(* IEC 61131-3 sources: sigmatek-logger-api/IXON_API/Class/cIXONConv10Value, 1 file *)

(* ---- cIXONConv10Value.st ---- *)
#DEFINE MAX_NAME_LENGTH 100
#DEFINE MAX_VALUE_LENGTH 10
#DEFINE MAX_DATASTRING_LENGTH 1024

(*!
<Class
	Name               = "cIXONConv10Value"
	Revision           = "0.0"
	RealtimeTask       = "false"
	CyclicTask         = "false"
	BackgroundTask     = "false"
	Sigmatek           = "false"
	OSInterface        = "false"
	HighPriority       = "false"
	Automatic          = "false"
	UpdateMode         = "Prescan"
	SharedCommandTable = "true"
	Objectsize         = "(510,120)">
	<Channels>
		<Server Name="ClassSvr" Visualized="false" Initialize="false" WriteProtected="true" Retentive="false"/>
		<Server Name="sCmdConvert" Visualized="false" Initialize="false" WriteProtected="false" Retentive="false"/>
		<Server Name="sName1" Class="String" Visualized="true" Initialize="true" WriteProtected="false" Retentive="false"/>
		<Server Name="sName10" Class="String" Visualized="true" Initialize="true" WriteProtected="false" Retentive="false"/>
		<Server Name="sName2" Class="String" Visualized="true" Initialize="true" WriteProtected="false" Retentive="false"/>
		<Server Name="sName3" Class="String" Visualized="true" Initialize="true" WriteProtected="false" Retentive="false"/>
		<Server Name="sName4" Class="String" Visualized="true" Initialize="true" WriteProtected="false" Retentive="false"/>
		<Server Name="sName5" Class="String" Visualized="true" Initialize="true" WriteProtected="false" Retentive="false"/>
		<Server Name="sName6" Class="String" Visualized="true" Initialize="true" WriteProtected="false" Retentive="false"/>
		<Server Name="sName7" Class="String" Visualized="true" Initialize="true" WriteProtected="false" Retentive="false"/>
		<Server Name="sName8" Class="String" Visualized="true" Initialize="true" WriteProtected="false" Retentive="false"/>
		<Server Name="sName9" Class="String" Visualized="true" Initialize="true" WriteProtected="false" Retentive="false"/>
		<Server Name="sSetInitNrOfEntrys" Visualized="false" Initialize="true" DefValue="1" WriteProtected="true" Retentive="false"/>
		<Server Name="sTriggerName" Class="String" Visualized="false" Initialize="true" WriteProtected="true" Retentive="false"/>
		<Server Name="sValue1" Visualized="false" Initialize="false" WriteProtected="false" Retentive="false"/>
		<Server Name="sValue10" Visualized="false" Initialize="false" WriteProtected="false" Retentive="false"/>
		<Server Name="sValue2" Visualized="false" Initialize="false" WriteProtected="false" Retentive="false"/>
		<Server Name="sValue3" Visualized="false" Initialize="false" WriteProtected="false" Retentive="false"/>
		<Server Name="sValue4" Visualized="false" Initialize="false" WriteProtected="false" Retentive="false"/>
		<Server Name="sValue5" Visualized="false" Initialize="false" WriteProtected="false" Retentive="false"/>
		<Server Name="sValue6" Visualized="false" Initialize="false" WriteProtected="false" Retentive="false"/>
		<Server Name="sValue7" Visualized="false" Initialize="false" WriteProtected="false" Retentive="false"/>
		<Server Name="sValue8" Visualized="false" Initialize="false" WriteProtected="false" Retentive="false"/>
		<Server Name="sValue9" Visualized="false" Initialize="false" WriteProtected="false" Retentive="false"/>
		<Client Name="Name1" Required="true" Internal="true"/>
		<Client Name="Name10" Required="true" Internal="true"/>
		<Client Name="Name2" Required="true" Internal="true"/>
		<Client Name="Name3" Required="true" Internal="true"/>
		<Client Name="Name4" Required="true" Internal="true"/>
		<Client Name="Name5" Required="true" Internal="true"/>
		<Client Name="Name6" Required="true" Internal="true"/>
		<Client Name="Name7" Required="true" Internal="true"/>
		<Client Name="Name8" Required="true" Internal="true"/>
		<Client Name="Name9" Required="true" Internal="true"/>
		<Client Name="ocSigCLib" Required="false" Internal="false"/>
		<Client Name="ToIXON_LoggerAPI" Required="true" Internal="false"/>
		<Client Name="TriggerName" Required="true" Internal="true"/>
	</Channels>
	<Separators>
		<Servers>
			<SepChn Position="3"/>
			<SepChn Position="5"/>
		</Servers>
	</Separators>
	<Network Name="cIXONConv10Value">
		<!-- List of Components in this network -->
		<Components>
			<Object
				Name       = "Name1"
				Class      = "String"
				Position   = "(420,300)"
				Visualized = "true"
				Remotely   = "true">
				<Channels>
					<Server Name="Data"/>
					<Client Name="SingleRealloc" Value="1"/>
				</Channels>
			</Object>
			<Object
				Name       = "Name10"
				Class      = "String"
				Position   = "(420,1650)"
				Visualized = "true"
				Remotely   = "true">
				<Channels>
					<Server Name="Data"/>
					<Client Name="SingleRealloc" Value="1"/>
				</Channels>
			</Object>
			<Object
				Name       = "Name2"
				Class      = "String"
				Position   = "(420,450)"
				Visualized = "true"
				Remotely   = "true">
				<Channels>
					<Server Name="Data"/>
					<Client Name="SingleRealloc" Value="1"/>
				</Channels>
			</Object>
			<Object
				Name       = "Name3"
				Class      = "String"
				Position   = "(420,600)"
				Visualized = "true"
				Remotely   = "true">
				<Channels>
					<Server Name="Data"/>
					<Client Name="SingleRealloc" Value="1"/>
				</Channels>
			</Object>
			<Object
				Name       = "Name4"
				Class      = "String"
				Position   = "(420,750)"
				Visualized = "true"
				Remotely   = "true">
				<Channels>
					<Server Name="Data"/>
					<Client Name="SingleRealloc" Value="1"/>
				</Channels>
			</Object>
			<Object
				Name       = "Name5"
				Class      = "String"
				Position   = "(420,900)"
				Visualized = "true"
				Remotely   = "true">
				<Channels>
					<Server Name="Data"/>
					<Client Name="SingleRealloc" Value="1"/>
				</Channels>
			</Object>
			<Object
				Name       = "Name6"
				Class      = "String"
				Position   = "(420,1050)"
				Visualized = "true"
				Remotely   = "true">
				<Channels>
					<Server Name="Data"/>
					<Client Name="SingleRealloc" Value="1"/>
				</Channels>
			</Object>
			<Object
				Name       = "Name7"
				Class      = "String"
				Position   = "(420,1200)"
				Visualized = "true"
				Remotely   = "true">
				<Channels>
					<Server Name="Data"/>
					<Client Name="SingleRealloc" Value="1"/>
				</Channels>
			</Object>
			<Object
				Name       = "Name8"
				Class      = "String"
				Position   = "(420,1350)"
				Visualized = "true"
				Remotely   = "true">
				<Channels>
					<Server Name="Data"/>
					<Client Name="SingleRealloc" Value="1"/>
				</Channels>
			</Object>
			<Object
				Name       = "Name9"
				Class      = "String"
				Position   = "(420,1500)"
				Visualized = "true"
				Remotely   = "true">
				<Channels>
					<Server Name="Data"/>
					<Client Name="SingleRealloc" Value="1"/>
				</Channels>
			</Object>
			<Object
				Name       = "TriggerName"
				Class      = "String"
				Position   = "(420,150)"
				Visualized = "true"
				Remotely   = "true">
				<Channels>
					<Server Name="Data"/>
					<Client Name="SingleRealloc" Value="1"/>
				</Channels>
			</Object>
		</Components>
		<Comments>
		</Comments>
		<!-- List of Connections in this network -->
		<Connections>
			<Connection Source="this.TriggerName" Destination="TriggerName.Data"/>
			<Connection Source="this.sTriggerName" Destination="TriggerName.Data" Vertices="(968,330),(796,240),"/>
			<Connection Source="this.Name1" Destination="Name1.Data"/>
			<Connection Source="this.sName1" Destination="Name1.Data" Vertices="(968,450),(796,390),"/>
			<Connection Source="this.Name2" Destination="Name2.Data"/>
			<Connection Source="this.sName2" Destination="Name2.Data" Vertices="(968,570),(796,540),"/>
			<Connection Source="this.Name3" Destination="Name3.Data"/>
			<Connection Source="this.Name4" Destination="Name4.Data"/>
			<Connection Source="this.Name5" Destination="Name5.Data"/>
			<Connection Source="this.sName3" Destination="Name3.Data" Vertices="(968,690),(796,690),"/>
			<Connection Source="this.sName4" Destination="Name4.Data" Vertices="(968,810),(796,840),"/>
			<Connection Source="this.Name6" Destination="Name6.Data"/>
			<Connection Source="this.Name7" Destination="Name7.Data"/>
			<Connection Source="this.sName5" Destination="Name5.Data" Vertices="(968,930),(796,990),"/>
			<Connection Source="this.sName6" Destination="Name6.Data" Vertices="(968,1050),(796,1140),"/>
			<Connection Source="this.sName7" Destination="Name7.Data" Vertices="(968,1170),(796,1290),"/>
			<Connection Source="this.Name8" Destination="Name8.Data"/>
			<Connection Source="this.Name9" Destination="Name9.Data"/>
			<Connection Source="this.Name10" Destination="Name10.Data"/>
			<Connection Source="this.sName8" Destination="Name8.Data" Vertices="(968,1290),(796,1440),"/>
			<Connection Source="this.sName9" Destination="Name9.Data" Vertices="(968,1410),(796,1590),"/>
			<Connection Source="this.sName10" Destination="Name10.Data" Vertices="(968,1530),(796,1740),"/>
		</Connections>
		<!-- Headerfiles -->
		<Options>
		</Options>
	</Network>
</Class>
*)
cIXONConv10Value : CLASS
  //Servers:
	ClassSvr 	: SvrChCmd_DINT;
	sSetInitNrOfEntrys 	: SvrCh_UDINT;
	sTriggerName 	: SvrChCmd_UDINT;
	sCmdConvert 	: SvrCh_DINT;
	sName1 	: SvrChCmd_UDINT;
	sValue1 	: SvrCh_DINT;
	sName2 	: SvrChCmd_UDINT;
	sValue2 	: SvrCh_DINT;
	sName3 	: SvrChCmd_UDINT;
	sValue3 	: SvrCh_DINT;
	sName4 	: SvrChCmd_UDINT;
	sValue4 	: SvrCh_DINT;
	sName5 	: SvrChCmd_UDINT;
	sValue5 	: SvrCh_DINT;
	sName6 	: SvrChCmd_UDINT;
	sValue6 	: SvrCh_DINT;
	sName7 	: SvrChCmd_UDINT;
	sValue7 	: SvrCh_DINT;
	sName8 	: SvrChCmd_UDINT;
	sValue8 	: SvrCh_DINT;
	sName9 	: SvrChCmd_UDINT;
	sValue9 	: SvrCh_DINT;
	sName10 	: SvrChCmd_UDINT;
	sValue10 	: SvrCh_DINT;
  //Clients:
	Name3 	: CltChCmd_String;
	Name2 	: CltChCmd_String;
	Name1 	: CltChCmd_String;
	Name4 	: CltChCmd_String;
	Name5 	: CltChCmd_String;
	Name6 	: CltChCmd_String;
	Name7 	: CltChCmd_String;
	Name8 	: CltChCmd_String;
	Name9 	: CltChCmd_String;
	Name10 	: CltChCmd_String;
	TriggerName 	: CltChCmd_String;
	ToIXON_LoggerAPI 	: CltChCmd_IXON_LoggerAPI_Interface;
	ocSigCLib 	: CltChCmd_SigCLib;
  //Variables:
		vNameString : ARRAY [0..MAX_NAME_LENGTH-1] OF CHAR;

		vValueString : ARRAY [0..MAX_VALUE_LENGTH-1] OF CHAR;

		vDataString : ARRAY [0..MAX_DATASTRING_LENGTH-1] OF CHAR;

  //Functions:

	FUNCTION BuildConfigString;

	FUNCTION BuildPair
		VAR_INPUT
			Value 	: DINT;
		END_VAR;

	FUNCTION BuildTrigger
		VAR_INPUT
			Value 	: DINT;
		END_VAR;

	FUNCTION VIRTUAL GLOBAL sTriggerName::Read
		VAR_OUTPUT
			output (EAX) 	: UDINT;
		END_VAR;

	FUNCTION VIRTUAL GLOBAL sTriggerName::Write
		VAR_INPUT
			input (EAX) 	: UDINT;
		END_VAR
		VAR_OUTPUT
			result (EAX) 	: UDINT;
		END_VAR;

	FUNCTION VIRTUAL GLOBAL sCmdConvert::Write
		VAR_INPUT
			input (EAX) 	: DINT;
		END_VAR
		VAR_OUTPUT
			result (EAX) 	: DINT;
		END_VAR;

	FUNCTION VIRTUAL GLOBAL sName1::Read
		VAR_OUTPUT
			output (EAX) 	: UDINT;
		END_VAR;

	FUNCTION VIRTUAL GLOBAL sName1::Write
		VAR_INPUT
			input (EAX) 	: UDINT;
		END_VAR
		VAR_OUTPUT
			result (EAX) 	: UDINT;
		END_VAR;

	FUNCTION VIRTUAL GLOBAL sName2::Read
		VAR_OUTPUT
			output (EAX) 	: UDINT;
		END_VAR;

	FUNCTION VIRTUAL GLOBAL sName2::Write
		VAR_INPUT
			input (EAX) 	: UDINT;
		END_VAR
		VAR_OUTPUT
			result (EAX) 	: UDINT;
		END_VAR;

	FUNCTION VIRTUAL GLOBAL sName3::Read
		VAR_OUTPUT
			output (EAX) 	: UDINT;
		END_VAR;

	FUNCTION VIRTUAL GLOBAL sName3::Write
		VAR_INPUT
			input (EAX) 	: UDINT;
		END_VAR
		VAR_OUTPUT
			result (EAX) 	: UDINT;
		END_VAR;

	FUNCTION VIRTUAL GLOBAL sName4::Read
		VAR_OUTPUT
			output (EAX) 	: UDINT;
		END_VAR;

	FUNCTION VIRTUAL GLOBAL sName4::Write
		VAR_INPUT
			input (EAX) 	: UDINT;
		END_VAR
		VAR_OUTPUT
			result (EAX) 	: UDINT;
		END_VAR;

	FUNCTION VIRTUAL GLOBAL sName5::Read
		VAR_OUTPUT
			output (EAX) 	: UDINT;
		END_VAR;

	FUNCTION VIRTUAL GLOBAL sName5::Write
		VAR_INPUT
			input (EAX) 	: UDINT;
		END_VAR
		VAR_OUTPUT
			result (EAX) 	: UDINT;
		END_VAR;

	FUNCTION VIRTUAL GLOBAL sName6::Read
		VAR_OUTPUT
			output (EAX) 	: UDINT;
		END_VAR;

	FUNCTION VIRTUAL GLOBAL sName6::Write
		VAR_INPUT
			input (EAX) 	: UDINT;
		END_VAR
		VAR_OUTPUT
			result (EAX) 	: UDINT;
		END_VAR;

	FUNCTION VIRTUAL GLOBAL sName7::Read
		VAR_OUTPUT
			output (EAX) 	: UDINT;
		END_VAR;

	FUNCTION VIRTUAL GLOBAL sName7::Write
		VAR_INPUT
			input (EAX) 	: UDINT;
		END_VAR
		VAR_OUTPUT
			result (EAX) 	: UDINT;
		END_VAR;

	FUNCTION VIRTUAL GLOBAL sName8::Read
		VAR_OUTPUT
			output (EAX) 	: UDINT;
		END_VAR;

	FUNCTION VIRTUAL GLOBAL sName8::Write
		VAR_INPUT
			input (EAX) 	: UDINT;
		END_VAR
		VAR_OUTPUT
			result (EAX) 	: UDINT;
		END_VAR;

	FUNCTION VIRTUAL GLOBAL sName9::Read
		VAR_OUTPUT
			output (EAX) 	: UDINT;
		END_VAR;

	FUNCTION VIRTUAL GLOBAL sName9::Write
		VAR_INPUT
			input (EAX) 	: UDINT;
		END_VAR
		VAR_OUTPUT
			result (EAX) 	: UDINT;
		END_VAR;

	FUNCTION VIRTUAL GLOBAL sName10::Read
		VAR_OUTPUT
			output (EAX) 	: UDINT;
		END_VAR;

	FUNCTION VIRTUAL GLOBAL sName10::Write
		VAR_INPUT
			input (EAX) 	: UDINT;
		END_VAR
		VAR_OUTPUT
			result (EAX) 	: UDINT;
		END_VAR;
  //Tables:
	FUNCTION @STD
		VAR_OUTPUT
			ret_code	: CONFSTATES;
		END_VAR;
	FUNCTION GLOBAL TAB @CT_;
END_CLASS;

#pragma using String
#pragma usingLtd IXON_LoggerAPI_Interface
#pragma usingLtd SigCLib

FUNCTION cIXONConv10Value::BuildConfigString
  VAR
    i : int;
    lValue : dint;
    length : udint;
  END_VAR

  if  sSetInitNrOfEntrys > 10
  then
      sSetInitNrOfEntrys := 10;
  end_if;

  _memset(dest:=#vDataString, usByte:=16#00, cntr:=MAX_DATASTRING_LENGTH);

  //Write trigger to 1 / true
  TriggerName.TxtGet(pdst :=  #vNameString[0], dstsize := sizeof(vNameString) - 1);
  BuildTrigger(Value := 1);

  //Setup JSON Object Pairs
  for i := 1  to to_int(sSetInitNrOfEntrys) do
    //Get Name
    case i of
      1: Name1.TxtGet(pdst := #vNameString[0], dstsize := sizeof(vNameString) - 1);
         lvalue := sValue1;
      2: Name2.TxtGet(pdst := #vNameString[0], dstsize := sizeof(vNameString) - 1);
         lvalue := sValue2;
      3: Name3.TxtGet(pdst := #vNameString[0], dstsize := sizeof(vNameString) - 1);
         lvalue := sValue3;
      4: Name4.TxtGet(pdst := #vNameString[0], dstsize := sizeof(vNameString) - 1);
         lvalue := sValue4;
      5: Name5.TxtGet(pdst := #vNameString[0], dstsize := sizeof(vNameString) - 1);
         lvalue := sValue5;
      6: Name6.TxtGet(pdst := #vNameString[0], dstsize := sizeof(vNameString) - 1);
         lvalue := sValue6;
      7: Name7.TxtGet(pdst := #vNameString[0], dstsize := sizeof(vNameString) - 1);
         lvalue := sValue7;
      8: Name8.TxtGet(pdst := #vNameString[0], dstsize := sizeof(vNameString) - 1);
         lvalue := sValue8;
      9: Name9.TxtGet(pdst := #vNameString[0], dstsize := sizeof(vNameString) - 1);
         lvalue := sValue9;
      10: Name10.TxtGet(pdst := #vNameString[0], dstsize := sizeof(vNameString) - 1);
         lvalue := sValue10;
    end_case;

    BuildPair(Value:=lValue);

  end_for;

  //Write trigger to 0 / false
  TriggerName.TxtGet(pdst :=  #vNameString[0], dstsize := sizeof(vNameString) - 1);
  BuildTrigger(Value := 0);

  length := _strlen(src:=#vDataString[0]);
  ToIXON_LoggerAPI.AddStringToBuffer(pData:=#vDataString[0], udLen:=length + 1);
END_FUNCTION

FUNCTION cIXONConv10Value::BuildPair
	VAR_INPUT
		Value 	: DINT;
	END_VAR
  VAR
  	length : UDINT;
  END_VAR

  ocSigCLib.IToA(val  := to_dint(Value),
                 dst  := #vValueString[0],
                 base := 10);

  length := _strlen(src:=#vDataString[0]);
  vDataString[length] := '@';
  _strcat(dest:=#vDataString[length + 1], src:=#vNameString[0]);
  length := _strlen(src:=#vDataString[0]);
  vDataString[length] := '=';
  _strcat(dest:=#vDataString[length + 1], src:=#vValueString[0]);
  length := _strlen(src:=#vDataString[0]);
  vDataString[length] := 16#0A;

END_FUNCTION

FUNCTION cIXONConv10Value::BuildTrigger
	VAR_INPUT
		Value 	: DINT;
	END_VAR
  VAR
  	length : UDINT;
  END_VAR

  ocSigCLib.IToA(val  := to_dint(Value),
                 dst  := #vValueString[0],
                 base := 10);

  length := _strlen(src:=#vDataString[0]);
  vDataString[length] := '@';
  _strcat(dest:=#vDataString[length + 1], src:=#vNameString[0]);
  length := _strlen(src:=#vDataString[0]);
  vDataString[length] := '=';
  if value = 0 then
    vDataString[length + 1] := 'f';
  else
    vDataString[length + 1] := 't';
  end_if;
  length := length + 2;
  vDataString[length] := 16#0A;

END_FUNCTION

FUNCTION VIRTUAL GLOBAL cIXONConv10Value::sCmdConvert::Write
	VAR_INPUT
		input (EAX) 	: DINT;
	END_VAR
	VAR_OUTPUT
		result (EAX) 	: DINT;
	END_VAR

	sCmdConvert := input;
	result := sCmdConvert;

  BuildConfigString();

END_FUNCTION

FUNCTION VIRTUAL GLOBAL cIXONConv10Value::sName1::Read
	VAR_OUTPUT
		output (EAX) 	: UDINT;
	END_VAR

	sName1 := Name1.Data.Read();
	output := sName1;

END_FUNCTION

FUNCTION VIRTUAL GLOBAL cIXONConv10Value::sName1::Write
	VAR_INPUT
		input (EAX) 	: UDINT;
	END_VAR
	VAR_OUTPUT
		result (EAX) 	: UDINT;
	END_VAR

	sName1 := input;
	result := (Name1.Data.Write(sName1))$UDINT;

END_FUNCTION

FUNCTION VIRTUAL GLOBAL cIXONConv10Value::sName2::Read
	VAR_OUTPUT
		output (EAX) 	: UDINT;
	END_VAR

	sName2 := Name2.Data.Read();
	output := sName2;

END_FUNCTION

FUNCTION VIRTUAL GLOBAL cIXONConv10Value::sName2::Write
	VAR_INPUT
		input (EAX) 	: UDINT;
	END_VAR
	VAR_OUTPUT
		result (EAX) 	: UDINT;
	END_VAR

	sName2 := input;
	result := (Name2.Data.Write(sName2))$UDINT;

END_FUNCTION

FUNCTION VIRTUAL GLOBAL cIXONConv10Value::sName3::Read
	VAR_OUTPUT
		output (EAX) 	: UDINT;
	END_VAR

	sName3 := Name3.Data.Read();
	output := sName3;

END_FUNCTION

FUNCTION VIRTUAL GLOBAL cIXONConv10Value::sName3::Write
	VAR_INPUT
		input (EAX) 	: UDINT;
	END_VAR
	VAR_OUTPUT
		result (EAX) 	: UDINT;
	END_VAR

	sName3 := input;
	result := (Name3.Data.Write(sName3))$UDINT;

END_FUNCTION

FUNCTION VIRTUAL GLOBAL cIXONConv10Value::sName4::Read
	VAR_OUTPUT
		output (EAX) 	: UDINT;
	END_VAR

	sName4 := Name4.Data.Read();
	output := sName4;

END_FUNCTION

FUNCTION VIRTUAL GLOBAL cIXONConv10Value::sName4::Write
	VAR_INPUT
		input (EAX) 	: UDINT;
	END_VAR
	VAR_OUTPUT
		result (EAX) 	: UDINT;
	END_VAR

	sName4 := input;
	result := (Name4.Data.Write(sName4))$UDINT;

END_FUNCTION

FUNCTION VIRTUAL GLOBAL cIXONConv10Value::sName5::Read
	VAR_OUTPUT
		output (EAX) 	: UDINT;
	END_VAR

	sName5 := Name5.Data.Read();
	output := sName5;

END_FUNCTION

FUNCTION VIRTUAL GLOBAL cIXONConv10Value::sName5::Write
	VAR_INPUT
		input (EAX) 	: UDINT;
	END_VAR
	VAR_OUTPUT
		result (EAX) 	: UDINT;
	END_VAR

	sName5 := input;
	result := (Name5.Data.Write(sName5))$UDINT;

END_FUNCTION

FUNCTION VIRTUAL GLOBAL cIXONConv10Value::sName6::Read
	VAR_OUTPUT
		output (EAX) 	: UDINT;
	END_VAR

	sName6 := Name6.Data.Read();
	output := sName6;

END_FUNCTION

FUNCTION VIRTUAL GLOBAL cIXONConv10Value::sName6::Write
	VAR_INPUT
		input (EAX) 	: UDINT;
	END_VAR
	VAR_OUTPUT
		result (EAX) 	: UDINT;
	END_VAR

	sName6 := input;
	result := (Name6.Data.Write(sName6))$UDINT;

END_FUNCTION

FUNCTION VIRTUAL GLOBAL cIXONConv10Value::sName7::Read
	VAR_OUTPUT
		output (EAX) 	: UDINT;
	END_VAR

	sName7 := Name7.Data.Read();
	output := sName7;

END_FUNCTION

FUNCTION VIRTUAL GLOBAL cIXONConv10Value::sName7::Write
	VAR_INPUT
		input (EAX) 	: UDINT;
	END_VAR
	VAR_OUTPUT
		result (EAX) 	: UDINT;
	END_VAR

	sName7 := input;
	result := (Name7.Data.Write(sName7))$UDINT;

END_FUNCTION

FUNCTION VIRTUAL GLOBAL cIXONConv10Value::sName8::Read
	VAR_OUTPUT
		output (EAX) 	: UDINT;
	END_VAR

	sName8 := Name8.Data.Read();
	output := sName8;

END_FUNCTION

FUNCTION VIRTUAL GLOBAL cIXONConv10Value::sName8::Write
	VAR_INPUT
		input (EAX) 	: UDINT;
	END_VAR
	VAR_OUTPUT
		result (EAX) 	: UDINT;
	END_VAR

	sName8 := input;
	result := (Name8.Data.Write(sName8))$UDINT;

END_FUNCTION

FUNCTION VIRTUAL GLOBAL cIXONConv10Value::sName9::Read
	VAR_OUTPUT
		output (EAX) 	: UDINT;
	END_VAR

	sName9 := Name9.Data.Read();
	output := sName9;

END_FUNCTION

FUNCTION VIRTUAL GLOBAL cIXONConv10Value::sName9::Write
	VAR_INPUT
		input (EAX) 	: UDINT;
	END_VAR
	VAR_OUTPUT
		result (EAX) 	: UDINT;
	END_VAR

	sName9 := input;
	result := (Name9.Data.Write(sName9))$UDINT;

END_FUNCTION

FUNCTION VIRTUAL GLOBAL cIXONConv10Value::sName10::Read
	VAR_OUTPUT
		output (EAX) 	: UDINT;
	END_VAR

	sName10 := Name10.Data.Read();
	output := sName10;

END_FUNCTION

FUNCTION VIRTUAL GLOBAL cIXONConv10Value::sName10::Write
	VAR_INPUT
		input (EAX) 	: UDINT;
	END_VAR
	VAR_OUTPUT
		result (EAX) 	: UDINT;
	END_VAR

	sName10 := input;
	result := (Name10.Data.Write(sName10))$UDINT;

END_FUNCTION

FUNCTION VIRTUAL GLOBAL cIXONConv10Value::sTriggerName::Read
	VAR_OUTPUT
		output (EAX) 	: UDINT;
	END_VAR

	sTriggerName := TriggerName.Data.Read();
	output := sTriggerName;

END_FUNCTION

FUNCTION VIRTUAL GLOBAL cIXONConv10Value::sTriggerName::Write
	VAR_INPUT
		input (EAX) 	: UDINT;
	END_VAR
	VAR_OUTPUT
		result (EAX) 	: UDINT;
	END_VAR

	sTriggerName := input;
	result := (TriggerName.Data.Write(sTriggerName))$UDINT;

END_FUNCTION
